FUNCTION IrDistanceFromRaw : REAL
VAR_INPUT
	rawValue : INT;
END_VAR
VAR
END_VAR

	//IrDistanceFromRaw := 123.15 / EXPT( INT_TO_REAL(rawValue) * (10.0 / 32767.0), 1.119 );

END_FUNCTION

(* stored: Version 1.1.0.1, ProductVersion 3.1.4024.11
   POU IrDistanceFromRaw: Id {5f98cdb0-3d47-495c-b636-8fc85b07fe47}, SpecialFunc None *)
